(* IEC 61131-3 sources: volt/packages/volt-lsp-iec/test-corpus/bakon-nano/Device/Plc Logic/Application/Library Manager/(unresolved)/systypes interfaces, 5 files *)

(* ---- RTS_IEC_CWCHAR.dut ---- *)
TYPE RTS_IEC_CWCHAR :
UNION
	WSNAME : WSTRING(255);
	SNAME : STRING(255);
END_UNION
END_TYPE

(* ---- RTS_IEC_HANDLE.dut ---- *)
TYPE RTS_IEC_HANDLE : POINTER TO BYTE;
END_TYPE

(* ---- RTS_IEC_RESULT.dut ---- *)
TYPE RTS_IEC_RESULT : UDINT;
END_TYPE

(* ---- RTS_IEC_SIZE.dut ---- *)
TYPE RTS_IEC_SIZE : POINTER TO BYTE;
END_TYPE

(* ---- HANDLECONSTANTS.gvl ---- *)
VAR_GLOBAL
	RTS_INVALID_HANDLE : RTS_IEC_HANDLE := -1;
END_VAR
